FUNCTION_BLOCK EL1052
VAR
	_io : EL1052_Data;
	{attribute addProperty Name "WcState"}
	_wcState : WcStateInputToggle;
	{attribute addProperty Name "Info data"}
	_infoData : InfoDataBase;
END_VAR

PROPERTY IO : REFERENCE TO EL1052_Data
GET
IO REF= _io;
END_GET
END_PROPERTY

PROPERTY WcState : REFERENCE TO WcStateInputToggle
GET
WcState REF= _wcState;
END_GET
END_PROPERTY

END_FUNCTION_BLOCK

(* stored: Version 1.1.0.1, ProductVersion 3.1.4024.9
   POU EL1052: Id {ae6f0455-d36a-0ecc-1d0f-eb6b8d0a25c5}, SpecialFunc None
   Property IO: Id {3a4882e9-2ad9-0d71-358e-800b502c9409}
   Get Get: Id {dded0e69-de51-07e9-1af9-3dc4dcc9e520}
   Property WcState: Id {56932313-6963-0787-3cb9-f1e95bd325b4}
   Get Get: Id {f68e60f2-2f0b-0866-24a5-c979f10c8b62} *)
